FUNCTION F_ITC_SendFSR : BOOL
(**************************************************************************************
 * 	Application		:	BoxControl Framework
 *	Revision		:	$Revision: 404529 $
 *	Revision date	:	$Date: 2018-04-23 08:21:38 +0200 (Mo., 23 Apr 2018) $
 *	Last changed by	:	$Author: b7bolm $
 *	URL				:	$URL: http://almscdc.swisslog.com/repo/SWPD/Development/BoxControlFramework/20_Release/trunk/01_Software/BCF/BCF/JumpStart/20_Product/10_App/11_Com/10_Lib/10_Conv/11_ITC/F_ITC_SendFSR.TcPOU $
 *
 *	Purpose			:	Wrap message - FSR
 *
 * ------------------------------------------------------------------------------------
 *	Copyright Swisslog [IP AG], Switzerland. All rights reserved.
 * 
 * ------------------------------------------------------------------------------------
 *	
 * 	Revision History: 
 *
 * 	VERSION			DATE			INITIALS			DESCRIPTION
 *	0.1				01.01.2001		swl					Example
 *
 **************************************************************************************)
VAR_INPUT
	eChannelSrc			: E_MFCS_Channel; // Source communicaton channel	
	FunctionName		: STRING(Conveyor.POSITION_STRINGLENGTH); // SIS MM-GGG-EEEE-FF-Z
	PrevFunctionNo		: STRING(Conveyor.POSITION_STRINGLENGTH); // SIS MM-GGG-EEEE-FF-Z
	NextFunctionNo		: STRING(Conveyor.POSITION_STRINGLENGTH); // SIS MM-GGG-EEEE-FF-Z
	eState				: E_PositionState; // State
	Enabled				: BOOL; // Enabled
	TransportState		: E_TransportState;
	TakeOverState		: E_TakeOverState;
	HandOverState		: E_HandOverState;
	TU_ID				: STRING(18); // 18 Digit SSID
	TU_Type				: INT; // TU Type
	AssignmentID		: UDINT; // Assignment ID
	LoadInformation		: INT; // 1 = Loaded, 0 = Not loaded
	Destination			: STRING(Conveyor.POSITION_STRINGLENGTH);
	eErrorState			: E_ErrorState; // Error State
	eErrorCode			: E_ErrorConv; // Return Code
	eErrorType			: E_ErrorType; // Error Type
	ErrorInformation	: STRING(System.ERROR_PARAM_STRINGLENGTH); // 5 Chars Error Information
	Variable			: DINT; // Variable
	eReturnCode			: E_ErrorConv; // Return code
END_VAR
VAR
	FSR					: ST_ITC_FSR; 
END_VAR

// Map values
FSR.Position			:= FunctionName;
FSR.PrevFunctionNo		:= PrevFunctionNo;
FSR.NextFunctionNo		:= NextFunctionNo;
FSR.eState				:= eState;
FSR.Enabled				:= Enabled;
FSR.TransportState		:= TransportState;
FSR.TakeOverState		:= TakeOverState;
FSR.HandOverState		:= HandOverState;
FSR.TU_ID				:= TU_ID;
FSR.TU_Type				:= TU_Type;
FSR.AssignmentID		:= AssignmentID;
FSR.LoadInformation		:= LoadInformation;
FSR.Destination			:= Destination;
FSR.eErrorState			:= eErrorState;
FSR.eErrorCode			:= eErrorCode;
FSR.eErrorType			:= eErrorType;
FSR.ErrorInformation	:= ErrorInformation;
FSR.Variable			:= Variable;
FSR.eReturnCode			:= eReturnCode;

// Forward to ITC
F_ITC_SendFSR := fbITC_Manager.M_SendData(
					meChannel	:= eChannelSrc,
					mMsgType	:= E_ITC_MsgTypeConv.FUNCTION_STATUS_REPORT,
					mpData		:= ADR(FSR),
					mLen		:= SIZEOF(FSR));

END_FUNCTION

(* stored: Version 1.1.0.1, ProductVersion 3.1.4022.12
   POU F_ITC_SendFSR: Id {b7d9265e-8f45-4905-a2e2-b12dba9db9ca}, SpecialFunc None *)
